PROGRAM MAIN
VAR
END_VAR

END_PROGRAM

(* stored: Version 1.1.0.1
   POU MAIN: Id {7032c09e-f7b2-48cc-90e2-d00191d9af4f} *)
